FUNCTION_BLOCK E_TOF (* standard timer function block (off-delay timing) *)
  (* Standard: 61499-2; Classification: standard timer function block; Description: Copyright (c) 2024 HR Agrartechnik GmbH This program and the accompanying materials are made available under the terms of the Eclipse Public License 2.0 which is available at https://www.eclipse.org/legal/epl-2.0/ SPDX-License-Identifier: EPL-2.0 E_TOF -- Off-delay timer FB When IN goes TRUE, Q becomes TRUE immediately. When IN goes FALSE, Q stays TRUE for duration PT before going FALSE. Reset stops the timer and sets Q to FALSE. *)
  (* Version 3.1, 2026-05-08, Franz Höpfinger, HR Agrartechnik GmbH, E_RF_TRIG instead of E_SWITCH *)
  (* Version 3.0, 2025-04-14, Patrick Aigner, changed package *)
  (* Version 1.1, 2024-04-23, Franz Höpfinger, HR Agrartechnik GmbH, Add a Reset to Timer FBs *)
  (* Version 1.0, 2024-03-04, Franz Höpfinger, HR Agrartechnik GmbH *)
  PACKAGE iec61499::events::timers;
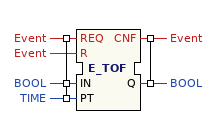
  EVENT_INPUT
    REQ WITH IN, PT; (* Normal Execution Request *)
    R; (* Reset *)
  END_EVENT
  EVENT_OUTPUT
    CNF WITH Q; (* Execution Confirmation *)
  END_EVENT
  VAR_INPUT
    IN : BOOL; (* Input *)
    PT : TIME; (* Process time *)
  END_VAR
  VAR_OUTPUT
    Q : BOOL; (* Output *)
  END_VAR
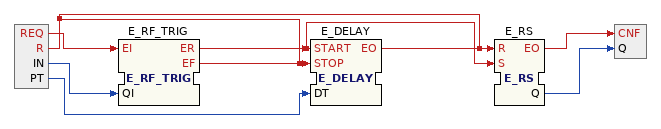
  FBS
    E_RF_TRIG : iec61499::events::E_RF_TRIG;
    E_DELAY : iec61499::events::E_DELAY;
    E_RS : iec61499::events::E_RS;
  END_FBS
  EVENT_CONNECTIONS
    REQ TO E_RF_TRIG.EI;
    E_RS.EO TO CNF;
    E_DELAY.EO TO E_RS.R;
    E_RF_TRIG.ER TO E_RS.S;
    E_RF_TRIG.ER TO E_DELAY.START;
    E_RF_TRIG.EF TO E_DELAY.STOP;
    R TO E_RS.R;
    R TO E_DELAY.STOP;
  END_CONNECTIONS
  DATA_CONNECTIONS
    IN TO E_RF_TRIG.QI;
    PT TO E_DELAY.DT;
    E_RS.Q TO Q;
  END_CONNECTIONS
END_FUNCTION_BLOCK
